// TIA Portal V19 export
VAR_GLOBAL   // PLC tag table "LB325"
   LB325_Pareggiatura_Pb_Aux2 AT %I302.1 : Bool;   // 356SH2
   LB325_Pareggiatura_Pb_Aux1 AT %I302.0 : Bool;   // 356SH1
   LB325_Pareggiatura_Lp_Aux2 AT %Q301.6 : Bool;   // 356SH2
   LB325_Pareggiatura_Lp_Aux1 AT %Q301.5 : Bool;   // 356SH1
END_VAR
